INTERFACE I_BoolArg EXTENDS I_Arg

PROPERTY Val : BOOL
GET
END_GET
END_PROPERTY

END_INTERFACE

(* stored: Version 1.1.0.1
   Itf I_BoolArg: Id {9d76ad8d-669f-4c52-a5c1-5fd937e33189}
   Property Val: Id {51afdc47-6de1-4749-a8ea-a48a77b384e6}
   Get Get: Id {60d0eac5-637f-4fca-8b41-b9fe686fbf72} *)
